// TIA Portal project "Andranik_voskanyan_PLC_project" (V20)

(* hardware
DEVICE "S7-1200 station_1"  S7-1200 Station
   slot 0: "Rack_0"  S7-1200 Rack  Rack  V1.0
   slot 1: "PLC_1"  CPU 1215C DC/DC/DC  6ES7 215-1AG40-0XB0  V4.6
*)

// ===== PLC "PLC_1"  CPU 1215C DC/DC/DC =====

VAR_GLOBAL   // PLC tag table "Default tag table"
   "emergencyButton" AT %I0.0 : Bool;
   "pedButtonDirB" AT %I0.1 : Bool;
   "pedButtonDirA" AT %I0.2 : Bool;
   "greenDirA" AT %Q0.0 : Bool;
   "yellowDirA" AT %Q0.1 : Bool;
   "redDirA" AT %Q0.2 : Bool;
   "pedGreenDirB" AT %Q0.3 : Bool;
   "pedRedDirB" AT %Q0.4 : Bool;
   "greenDirB" AT %Q0.5 : Bool;
   "yellowDirB" AT %Q0.6 : Bool;
   "redDirB" AT %Q0.7 : Bool;
   "pedGreenDirA" AT %Q1.0 : Bool;
   "pedRedDirA" AT %Q1.1 : Bool;
   "Tag_1" AT %M0.0 : Bool;
   "Tag_2" AT %M0.1 : Bool;
   "Tag_3" AT %M0.2 : Bool;
   "Tag_4" AT %M0.3 : Bool;
   "Tag_5" AT %M0.5 : Bool;
   "Tag_7" AT %M1.0 : Bool;
   "Tag_8" AT %M1.1 : Bool;
   "Tag_9" AT %M2.1 : Bool;
   "Tag_10" AT %M2.2 : Bool;
   "Tag_11" AT %M2.3 : Bool;
   "Tag_12" AT %M1.2 : Bool;
   "Tag_13" AT %M3.0 : Bool;
   "Tag_14" AT %M4.0 : Bool;
   "Tag_15" AT %M3.1 : Bool;
   "Tag_16" AT %M3.2 : Bool;
   "Tag_17" AT %M4.1 : Bool;
   "Tag_18" AT %M3.3 : Bool;
   "Tag_19" AT %M3.4 : Bool;
   "Tag_20" AT %M3.5 : Bool;
   "Tag_21" AT %M2.4 : Bool;
   "Tag_22" AT %M4.2 : Bool;
   "Tag_23" AT %M4.3 : Bool;
   "start" AT %M0.7 : Bool;
   "reset" AT %M0.6 : Bool;
END_VAR

// folder: System blocks/Program resources

DATA_BLOCK "IEC_Timer_0_DB_1"   // DB2
{ S7_Optimized_Access := 'TRUE' }
AUTHOR : Simatic
FAMILY : IEC
NAME : IEC_TMR
VERSION : 1.0
// stored: InstanceOfName IEC_TIMER
"IEC_TIMER"
BEGIN
END_DATA_BLOCK

DATA_BLOCK "IEC_Timer_0_DB_2"   // DB3
{ S7_Optimized_Access := 'TRUE' }
AUTHOR : Simatic
FAMILY : IEC
NAME : IEC_TMR
VERSION : 1.0
// stored: InstanceOfName IEC_TIMER
"IEC_TIMER"
BEGIN
END_DATA_BLOCK

DATA_BLOCK "IEC_Timer_0_DB_3"   // DB4
{ S7_Optimized_Access := 'TRUE' }
AUTHOR : Simatic
FAMILY : IEC
NAME : IEC_TMR
VERSION : 1.0
// stored: InstanceOfName IEC_TIMER
"IEC_TIMER"
BEGIN
END_DATA_BLOCK

DATA_BLOCK "IEC_Timer_0_DB_4"   // DB5
{ S7_Optimized_Access := 'TRUE' }
AUTHOR : Simatic
FAMILY : IEC
NAME : IEC_TMR
VERSION : 1.0
// stored: InstanceOfName IEC_TIMER
"IEC_TIMER"
BEGIN
END_DATA_BLOCK

DATA_BLOCK "IEC_Timer_0_DB_5"   // DB6
{ S7_Optimized_Access := 'TRUE' }
AUTHOR : Simatic
FAMILY : IEC
NAME : IEC_TMR
VERSION : 1.0
// stored: InstanceOfName IEC_TIMER
"IEC_TIMER"
BEGIN
END_DATA_BLOCK

DATA_BLOCK "IEC_Timer_0_DB_6"   // DB7
{ S7_Optimized_Access := 'TRUE' }
AUTHOR : Simatic
FAMILY : IEC
NAME : IEC_TMR
VERSION : 1.0
// stored: InstanceOfName IEC_TIMER
"IEC_TIMER"
BEGIN
END_DATA_BLOCK

// folder: (top level)

FUNCTION "Push_on_push_off" : Void   // FC1, LAD
{ S7_Optimized_Access := 'TRUE' }
VERSION : 0.1
   VAR_INPUT
      button : Bool;
   END_VAR
   VAR_IN_OUT
      out : Bool;
      stage1 : Bool;
      stage2 : Bool;
   END_VAR
BEGIN

REGION Network 1
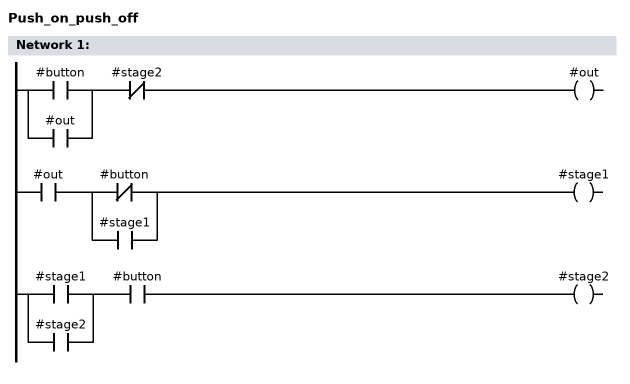
   RUNG wire#powerrail
      Contact( #button )
      wire#w1
      I_Contact( #stage2 )
      Coil( #out )
   END_RUNG
   RUNG wire#powerrail
      Contact( #out )
   END_RUNG wire#w1
   RUNG wire#powerrail
      Contact( #out )
      wire#w2
      I_Contact( #button )
      wire#w3
      Coil( #stage1 )
   END_RUNG
   RUNG wire#w2
      Contact( #stage1 )
   END_RUNG wire#w3
   RUNG wire#powerrail
      Contact( #stage1 )
      wire#w4
      Contact( #button )
      Coil( #stage2 )
   END_RUNG
   RUNG wire#powerrail
      Contact( #stage2 )
   END_RUNG wire#w4
   // the same network as SCL:
   #out := (#button OR #out) AND NOT #stage2;
   #stage1 := #out AND (NOT #button OR #stage1);
   #stage2 := (#stage1 OR #stage2) AND #button;
END_REGION
END_FUNCTION

ORGANIZATION_BLOCK "Main"   // OB1, LAD, ProgramCycle
TITLE = "Main Program Sweep (Cycle)"
{ S7_Optimized_Access := 'TRUE' }
VERSION : 0.1
   VAR_INPUT
      Initial_Call : Bool;   // Initial call of this OB
      Remanence : Bool;   // =True, if remanent data are available
   END_VAR
   VAR_TEMP   // added for the SCL form of the ladder/FBD networks
      _w1 : Bool;
      _w2 : Bool;
      _w3 : Bool;
      _w4 : Bool;
      _w5 : Bool;
      _w6 : Bool;
   END_VAR
BEGIN

REGION Network 1
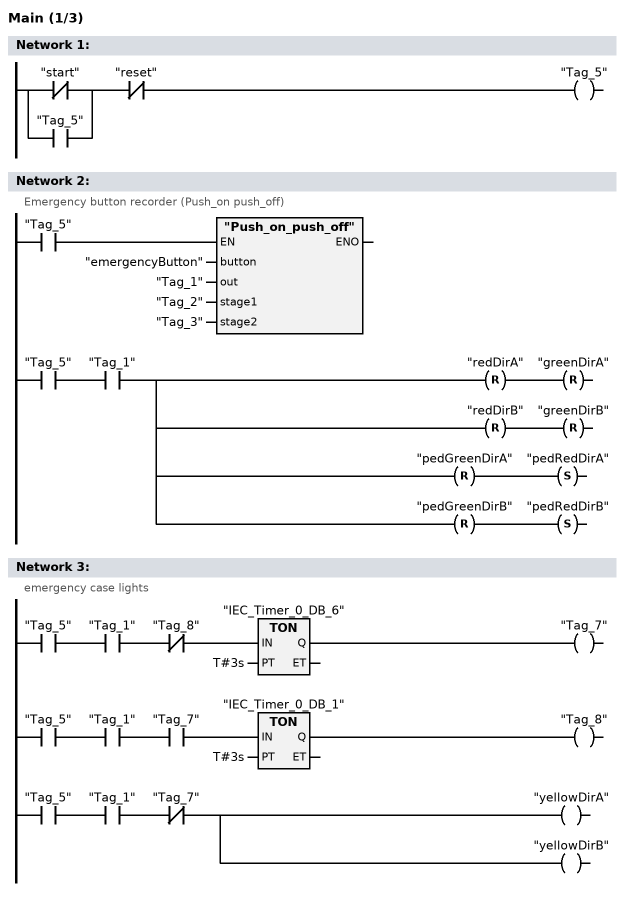
   RUNG wire#powerrail
      I_Contact( "start" )
      wire#w1
      I_Contact( "reset" )
      Coil( "Tag_5" )
   END_RUNG
   RUNG wire#powerrail
      Contact( "Tag_5" )
   END_RUNG wire#w1
   // the same network as SCL:
   "Tag_5" := (NOT "start" OR "Tag_5") AND NOT "reset";
END_REGION

REGION Network 2
   // Emergency button recorder (Push_on push_off)
   RUNG wire#powerrail
      Contact( "Tag_5" )
      "Push_on_push_off"(button := "emergencyButton", out := "Tag_1", stage1 := "Tag_2", stage2 := "Tag_3")
   END_RUNG
   RUNG wire#powerrail
      Contact( "Tag_5" )
      Contact( "Tag_1" )
      wire#w1
      R_Coil( "redDirA" )
      R_Coil( "greenDirA" )
   END_RUNG
   RUNG wire#w1
      R_Coil( "redDirB" )
      R_Coil( "greenDirB" )
   END_RUNG
   RUNG wire#w1
      R_Coil( "pedGreenDirA" )
      S_Coil( "pedRedDirA" )
   END_RUNG
   RUNG wire#w1
      R_Coil( "pedGreenDirB" )
      S_Coil( "pedRedDirB" )
   END_RUNG
   // the same network as SCL:
   IF "Tag_5" THEN
       "Push_on_push_off"(button := "emergencyButton", out := "Tag_1", stage1 := "Tag_2", stage2 := "Tag_3");
   END_IF;
   IF "Tag_5" AND "Tag_1" THEN
       "redDirA" := FALSE;
       "greenDirA" := FALSE;
       "redDirB" := FALSE;
       "greenDirB" := FALSE;
       "pedGreenDirA" := FALSE;
       "pedRedDirA" := TRUE;
       "pedGreenDirB" := FALSE;
       "pedRedDirB" := TRUE;
   END_IF;
END_REGION

REGION Network 3
   // emergency case lights
   "IEC_Timer_0_DB_6".TON(IN := "Tag_5" AND "Tag_1" AND NOT "Tag_8", PT := T#3s);
   "Tag_7" := "IEC_Timer_0_DB_6".Q;
   "IEC_Timer_0_DB_1".TON(IN := "Tag_5" AND "Tag_1" AND "Tag_7", PT := T#3s);
   "Tag_8" := "IEC_Timer_0_DB_1".Q;
   "yellowDirA" := "Tag_5" AND "Tag_1" AND NOT "Tag_7";
   "yellowDirB" := "yellowDirA";
END_REGION

REGION Network 4
   // light without emergancy
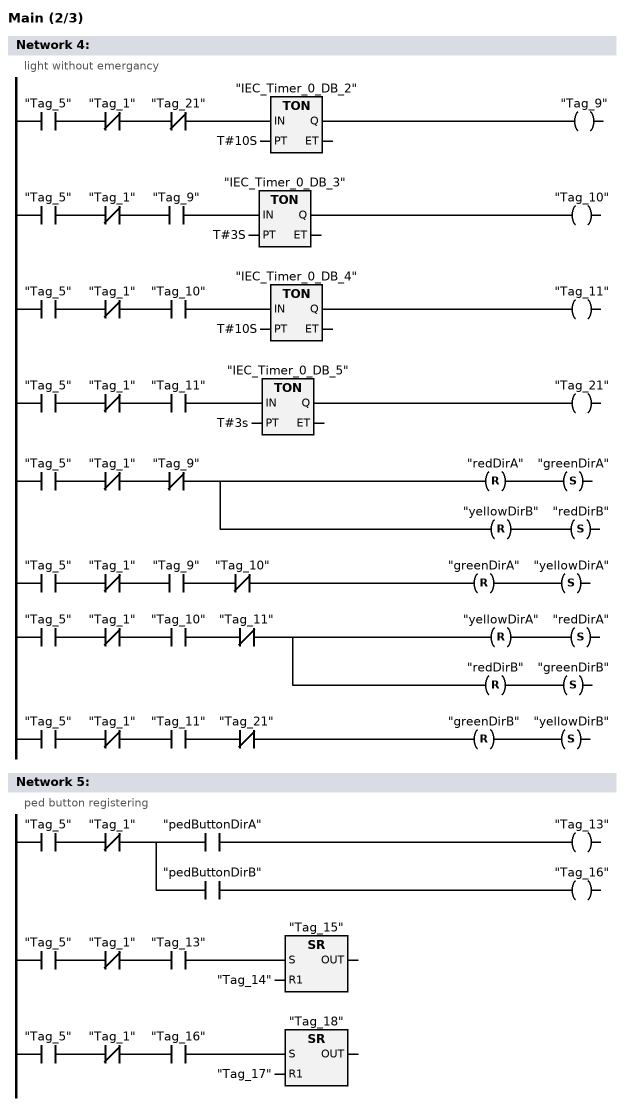
   "IEC_Timer_0_DB_2".TON(IN := "Tag_5" AND NOT "Tag_1" AND NOT "Tag_21", PT := T#10S);
   "Tag_9" := "IEC_Timer_0_DB_2".Q;
   "IEC_Timer_0_DB_3".TON(IN := "Tag_5" AND NOT "Tag_1" AND "Tag_9", PT := T#3S);
   "Tag_10" := "IEC_Timer_0_DB_3".Q;
   "IEC_Timer_0_DB_4".TON(IN := "Tag_5" AND NOT "Tag_1" AND "Tag_10", PT := T#10S);
   "Tag_11" := "IEC_Timer_0_DB_4".Q;
   "IEC_Timer_0_DB_5".TON(IN := "Tag_5" AND NOT "Tag_1" AND "Tag_11", PT := T#3s);
   "Tag_21" := "IEC_Timer_0_DB_5".Q;
   IF "Tag_5" AND NOT "Tag_1" AND NOT "Tag_9" THEN
       "redDirA" := FALSE;
       "greenDirA" := TRUE;
       "yellowDirB" := FALSE;
       "redDirB" := TRUE;
   END_IF;
   IF "Tag_5" AND NOT "Tag_1" AND "Tag_9" AND NOT "Tag_10" THEN
       "greenDirA" := FALSE;
       "yellowDirA" := TRUE;
   END_IF;
   IF "Tag_5" AND NOT "Tag_1" AND "Tag_10" AND NOT "Tag_11" THEN
       "yellowDirA" := FALSE;
       "redDirA" := TRUE;
       "redDirB" := FALSE;
       "greenDirB" := TRUE;
   END_IF;
   IF "Tag_5" AND NOT "Tag_1" AND "Tag_11" AND NOT "Tag_21" THEN
       "greenDirB" := FALSE;
       "yellowDirB" := TRUE;
   END_IF;
END_REGION

REGION Network 5
   // ped button registering
   RUNG wire#powerrail
      Contact( "Tag_5" )
      I_Contact( "Tag_1" )
      wire#w1
      Contact( "pedButtonDirA" )
      Coil( "Tag_13" )
   END_RUNG
   RUNG wire#w1
      Contact( "pedButtonDirB" )
      Coil( "Tag_16" )
   END_RUNG
   RUNG wire#powerrail
      Contact( "Tag_5" )
      I_Contact( "Tag_1" )
      Contact( "Tag_13" )
      S_SR(operand := "Tag_15", r1 := "Tag_14")
   END_RUNG
   RUNG wire#powerrail
      Contact( "Tag_5" )
      I_Contact( "Tag_1" )
      Contact( "Tag_16" )
      S_SR(operand := "Tag_18", r1 := "Tag_17")
   END_RUNG
   // the same network as SCL:
   #_w1 := "Tag_5" AND NOT "Tag_1";
   "Tag_13" := #_w1 AND "pedButtonDirA";
   "Tag_16" := #_w1 AND "pedButtonDirB";
   IF "Tag_5" AND NOT "Tag_1" AND "Tag_13" THEN
       "Tag_15" := TRUE;   // SR flip-flop
   END_IF;
   IF "Tag_14" THEN "Tag_15" := FALSE; END_IF;
   IF "Tag_5" AND NOT "Tag_1" AND "Tag_16" THEN
       "Tag_18" := TRUE;   // SR flip-flop
   END_IF;
   IF "Tag_17" THEN "Tag_18" := FALSE; END_IF;
END_REGION

REGION Network 6
   // lights of pedestrian
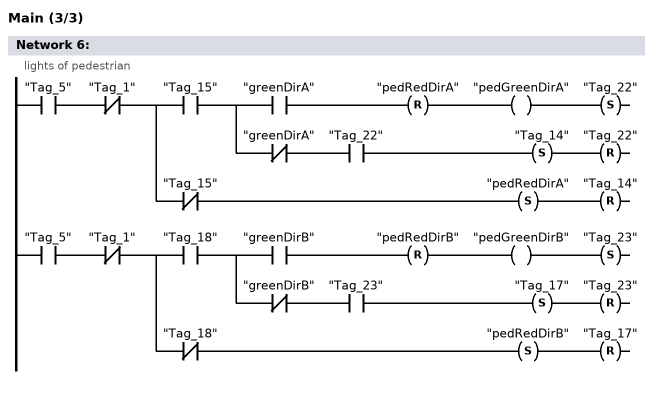
   RUNG wire#powerrail
      Contact( "Tag_5" )
      I_Contact( "Tag_1" )
      wire#w1
      Contact( "Tag_15" )
      wire#w2
      Contact( "greenDirA" )
      R_Coil( "pedRedDirA" )
      Coil( "pedGreenDirA" )
      S_Coil( "Tag_22" )
   END_RUNG
   RUNG wire#w2
      I_Contact( "greenDirA" )
      Contact( "Tag_22" )
      S_Coil( "Tag_14" )
      R_Coil( "Tag_22" )
   END_RUNG
   RUNG wire#w1
      I_Contact( "Tag_15" )
      S_Coil( "pedRedDirA" )
      R_Coil( "Tag_14" )
   END_RUNG
   RUNG wire#powerrail
      Contact( "Tag_5" )
      I_Contact( "Tag_1" )
      wire#w3
      Contact( "Tag_18" )
      wire#w4
      Contact( "greenDirB" )
      R_Coil( "pedRedDirB" )
      Coil( "pedGreenDirB" )
      S_Coil( "Tag_23" )
   END_RUNG
   RUNG wire#w4
      I_Contact( "greenDirB" )
      Contact( "Tag_23" )
      S_Coil( "Tag_17" )
      R_Coil( "Tag_23" )
   END_RUNG
   RUNG wire#w3
      I_Contact( "Tag_18" )
      S_Coil( "pedRedDirB" )
      R_Coil( "Tag_17" )
   END_RUNG
   // the same network as SCL:
   #_w1 := "Tag_5" AND NOT "Tag_1";
   #_w2 := #_w1 AND "Tag_15";
   #_w3 := #_w2 AND "greenDirA";
   IF #_w3 THEN "pedRedDirA" := FALSE; END_IF;
   "pedGreenDirA" := #_w3;
   IF #_w3 THEN "Tag_22" := TRUE; END_IF;
   IF #_w2 AND NOT "greenDirA" AND "Tag_22" THEN
       "Tag_14" := TRUE;
       "Tag_22" := FALSE;
   END_IF;
   IF #_w1 AND NOT "Tag_15" THEN
       "pedRedDirA" := TRUE;
       "Tag_14" := FALSE;
   END_IF;
   #_w4 := "Tag_5" AND NOT "Tag_1";
   #_w5 := #_w4 AND "Tag_18";
   #_w6 := #_w5 AND "greenDirB";
   IF #_w6 THEN "pedRedDirB" := FALSE; END_IF;
   "pedGreenDirB" := #_w6;
   IF #_w6 THEN "Tag_23" := TRUE; END_IF;
   IF #_w5 AND NOT "greenDirB" AND "Tag_23" THEN
       "Tag_17" := TRUE;
       "Tag_23" := FALSE;
   END_IF;
   IF #_w4 AND NOT "Tag_18" THEN
       "pedRedDirB" := TRUE;
       "Tag_17" := FALSE;
   END_IF;
END_REGION
END_ORGANIZATION_BLOCK